// TwinCAT 3 PLC project Untitled1
// ProgramVersion: 3.1.4022.2
// libraries:
//   Tc2_EtherCAT, * (Beckhoff Automation GmbH)
//   Tc2_Standard, * (Beckhoff Automation GmbH)
//   Tc2_System, * (Beckhoff Automation GmbH)
//   Tc2_Utilities, * (Beckhoff Automation GmbH)
//   Tc3_Module, * (Beckhoff Automation GmbH)
//   VisuSymbols,3.5.10.0,System
// project tree:
//   / GlobalTextList.TcGTLO, PlcTask.TcTTO, Visualization Manager.TcVMO (not stored)
//   POUs/ MAIN.TcPOU, STRING_BUFFER.TcPOU
//   VISUs/ Visualization.TcVIS
// real-time tasks:
//   TASK PlcTask: cycle T#100us, priority 20, ADS port 350
//   TASK VISU_TASK: cycle T#200000us, priority 30, ADS port 351
// I/O:
//   DEVICE Device 1 (EtherCAT), AmsNetId 5.49.22.42.2.1
//     Term 1 (EK1200) [EK1200-5000 EtherCAT Power supply (2A E-Bus)]
//       Term 2 (EL5101) [EL5101 1Ch. Inc. Encoder 5V]
//       Term 3 (EL9011) [EL9011 End Terminal]
// variable links:
//   Untitled1 Instance <-> Device 1 (EtherCAT)/Term 1 (EK1200)/Term 2 (EL5101)
//     PlcTask Inputs/MAIN.enc_raw <-> ENC Status compact/Counter value

CONFIGURATION Untitled1
    RESOURCE PLC ON TwinCAT3
        TASK PlcTask(INTERVAL := T#100us, PRIORITY := 20);
        PROGRAM MAIN WITH PlcTask : MAIN;
    END_RESOURCE
END_CONFIGURATION

// ---- POUs/MAIN.TcPOU
PROGRAM MAIN
VAR
	heartbeat 		: UDINT;
	
	enc_raw AT %I* 	: UINT;
	enc_angle 		: REAL;
	
	// Time
	tDC 			: T_DCTIME64;
	sTime 			: STRING;
	
	// File writing
	bRecordData 	: BOOL;
	iFileState 		: UINT;
	sFilePath 		: STRING 	:= 'C:\Users\Public\Documents\EncoderData\test.csv';
	fbRecordTrigger	: R_TRIG;
	
	fbFileOpen		: FB_FileOpen; 				// Opens file
	fbFileClose		: FB_FileClose;				// Closes file
	fbFileWriter		: FB_FileWrite;			// Writes binary
	
	sLineToWrite	: STRING;
	
	bBusy			: BOOL;
	bError			: BOOL;
	nErrId			: UDINT;
	hFile			: UINT		:= 0;
	
	iStartWrite		: UDINT;					// PLC scans at start of write
	iWriteScans		: UDINT;					// PLC scans between writes
	
	// Buffer
	sBuffer 		: ARRAY [0..iBufferLength] OF STRING;
	sLineToBuffer	: STRING;
	cbCurrentBufferLength : UDINT;
	sBufferToWrite	: ARRAY [0..iBufferLength] OF STRING;
	bBufferFull 	: BOOL;
	
END_VAR
VAR CONSTANT
	iBufferLength	: UDINT		:= 50;
	iLineLength 	: UDINT		:= 24;
END_VAR

heartbeat := heartbeat + 1;

enc_angle := enc_raw MOD (360*4);
enc_angle := enc_angle / 4;

tDC := F_GetCurDcTaskTime64();
sTime := DCTIME64_TO_STRING(tDC);

fbRecordTrigger(CLK:=bRecordData);
IF fbRecordTrigger.Q THEN
	// Clear the buffer when we start recording
	MEMSET( destAddr := ADR(sBuffer),
			fillByte := 0,
			n := iLineLength * iBufferLength);
	cbCurrentBufferLength := 0;
END_IF

IF bRecordData AND NOT bBufferFull THEN
	// Prepare the line to buffer
	sLineToBuffer := '';
	sLineToBuffer := CONCAT(ULINT_TO_STRING(tDC), ', ');
	sLineToBuffer := CONCAT(sLineToBuffer, UINT_TO_STRING(enc_raw));
	sLineToBuffer := CONCAT(sLineToBuffer, '$L');

	// Copy the line into the buffer
	MEMCPY(	srcAddr := ADR(sLineToBuffer),
			destAddr := ADR(sBuffer) + cbCurrentBufferLength * iLineLength,
			n := iLineLength);
	
	cbCurrentBufferLength := cbCurrentBufferLength + 1;
END_IF

IF iBufferLength > cbCurrentBufferLength THEN
	bBufferFull := FALSE;
ELSE
	bBufferFull := TRUE;
END_IF

CASE iFileState OF
	0:	// Wait to start
		IF bRecordData THEN
			bBusy := TRUE;
			
			// Reset some variables
			bError	:= FALSE;
			nErrId	:= 0;
			hFile	:= 0;
			
			iFileState := 10;
		END_IF
		
	10:	// Open the file
		fbFileOpen(bExecute := FALSE);
		fbFileOpen(	sNetId := '', 
					sPathName := sFilePath, 
					nMode := FOPEN_MODEWRITE OR FOPEN_MODEBINARY, 
					ePath := PATH_GENERIC, 
					bExecute := TRUE);
		iFileState := 20;
	
	20:	// Wait for opening to finish
		fbFileOpen(bExecute := FALSE, bError => bError, nErrID => nErrID, hFile => hFile );
		IF NOT fbFileOpen.bBusy THEN
			IF NOT fbFileOpen.bError THEN
				iFileState := 30;
			ELSE(* Error: file not found? *)
				iFileState := 100;
			END_IF
		END_IF
		
	30: // If we still want to write the file, write it
		IF bRecordData THEN
			// Clear the writer's buffer						
			MEMSET( destAddr := ADR(sBufferToWrite),
					fillByte := 0,
					n := iLineLength * iBufferLength);
		
			MEMCPY(	srcAddr := ADR(sBuffer),
					destAddr := ADR(sBufferToWrite),
					n := cbCurrentBufferLength * iLineLength);
			
			fbFileWriter( sNetId := '',
						hFile := hFile,
						pWriteBuff := ADR(sBufferToWrite),
						cbWriteLen := cbCurrentBufferLength * iLineLength,
						bExecute := TRUE);
			
			// Clear the buffer						
			MEMSET( destAddr := ADR(sBuffer),
					fillByte := 0,
					n := iLineLength * iBufferLength);
			cbCurrentBufferLength := 0;
						
			iWriteScans := heartbeat - iStartWrite;
			iStartWrite := heartbeat;
			
			iFileState := 40;
		
		ELSE // Stop writing
			iFileState := 200;
		END_IF
		
	40:	// Wait for the write to finish
		fbFileWriter( bExecute := FALSE, bError => bError, nErrID => nErrID );
		IF NOT fbFileWriter.bBusy THEN
			IF NOT fbFileWriter.bError THEN
				iFileState := 30;(* Write next record *)
			ELSE(* Error *)
				iFileState := 100;
			END_IF
		END_IF
			
	100: // Error
		IF ( hFile <> 0 ) THEN
			iFileState := 200; (* Close the source file *)
		ELSE
			bBusy := FALSE;
			iFileState := 0;	(* Ready *)
		END_IF
		
	200: // Close
		fbFileClose( bExecute := FALSE );
		fbFileClose( sNetId := '', hFile := hFile, bExecute := TRUE );
		iFileState := 210;
		
	210: // Wait for close to finish
		fbFileClose( bExecute := FALSE, bError => bError, nErrID => nErrID );
		IF ( NOT fbFileClose.bBusy ) THEN
			hFile := 0;
			bBusy := FALSE;
			iFileState := 0;	(* Ready *)
		END_IF

END_CASE

END_PROGRAM

// ---- POUs/STRING_BUFFER.TcPOU
FUNCTION_BLOCK STRING_BUFFER
VAR CONSTANT
	iBufferLength : UINT := 50;
END_VAR
VAR_INPUT
	
END_VAR
VAR_OUTPUT
END_VAR
VAR
END_VAR

END_FUNCTION_BLOCK

// ---- GlobalTextList.TcGTLO
TEXTLIST GlobalTextList
  936 = 'iFileState: %d'
  685 = 'Recording? %s'
  113 = 'Write'
END_TEXTLIST

// ---- VISUs/Visualization.TcVIS
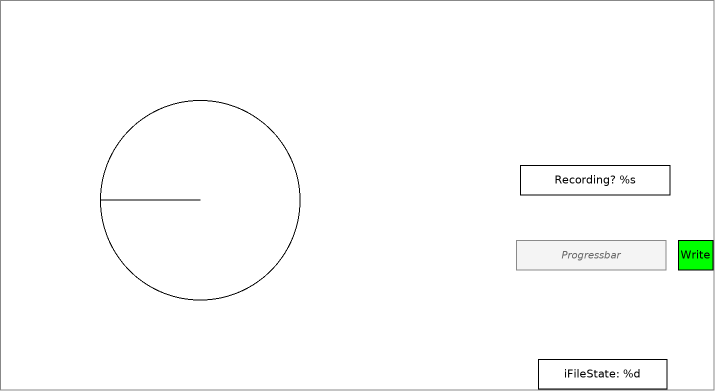
VISUALIZATION Visualization  // 715x391
    Rectangle (520,165 150x30), "Recording? %s", text variable: MAIN.bRecordData
        OnMouseDown: execute { MAIN.bRecordData := NOT MAIN.bRecordData; }
    Ellipse (100,100 200x200)
    Line (200,200) (100,200)
        p2858320360: MAIN.enc_angle
    Progressbar (516,240 150x30), variable: MAIN.cbCurrentBufferLength
    Rectangle (678,240 35x30), "Write", text variable: MAIN.bRecordData, invisible if: not MAIN.fbFileWriter.bBusy
    Rectangle (538,359 129x30), "iFileState: %d", text variable: MAIN.iFileState
END_VISUALIZATION
